PROGRAM Hardware
VAR
END_VAR

END_PROGRAM

(* stored: Version 1.1.0.1, ProductVersion 3.1.4024.13
   POU Hardware: Id {7c48af90-6723-4880-a33e-8559ccab70bd}, SpecialFunc None *)
